// TIA Portal V20 export
// export: Created 2025-12-01T14:57:23.6225211Z, ExportSetting None, DisplayName Totally Integrated Automation Portal, DisplayVersion V20 Update 3, DisplayName TIA Portal Openness, DisplayVersion V20 Update 3, DisplayName TIA Portal Version Control Interface, DisplayVersion V20 Update 3, DisplayName STEP 7 Professional, DisplayVersion V20 Update 3, DisplayName STEP 7 Safety, DisplayVersion V20 Update 2, DisplayName WinCC Basic/Comfort/Advanced, DisplayVersion V20 Update 3, DisplayName WinCC Professional, DisplayVersion V20 Update 3, DisplayName WinCC Unified, DisplayVersion V20 Update 3
DATA_BLOCK "DB010_ScadaConfig"   // DB10
{ S7_Optimized_Access := 'FALSE' }
AUTHOR : SCADA
NAME : 20161001
VERSION : 1.0
// stored: AutoNumber false
   VAR RETAIN
      NDB_ScadaZona : Int := 13;   // Datos del DB 13 (DB PLC ==> SCADA)
      Long_ScadaZona : Int := 24;
      OffEstado_ScadaZona : Int := 0;
      OffCodigo_ScadaZona : Int := 2;
      OffEntrada_ScadaZona : Int := 6;
      OffSalida_ScadaZona : Int := 8;
      OffDatos_ScadaZona : Int := 10;
      OffEmergGrave_ScadaZona : Int := 12;
      OffEmergLeve_ScadaZona : Int := 14;
      OffErrGrave_ScadaZona : Int := 18;
      OffErrLeve_ScadaZona : Int := 20;
   END_VAR
BEGIN
END_DATA_BLOCK
